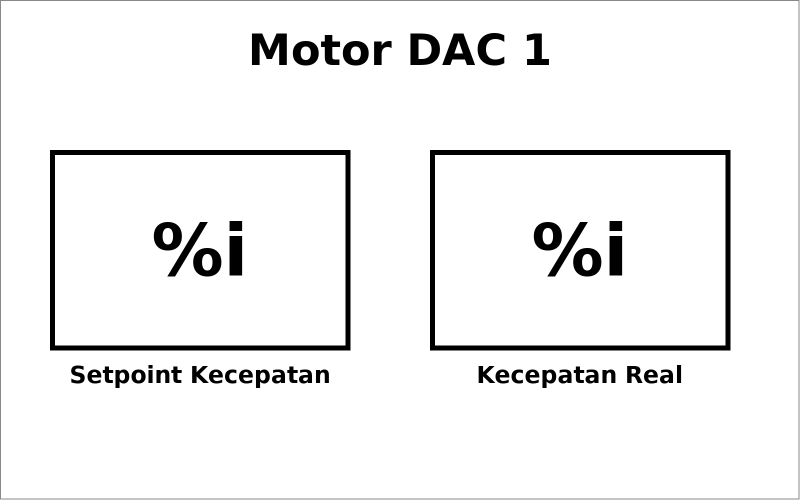
VISUALIZATION Screen_2_Sub_2  // 800x500
    Label (0,0 800x100), "Motor DAC 1"
    Rectangle (50,150 300x200), "%i", text variable: GVL.HMI_Motor_DAC_1_Input
        OnMouseClick: write GVL.HMI_Motor_DAC_1_Input via VisuDialogs.Numpad
    Label (50,350 300x50), "Setpoint Kecepatan"
    Label (430,350 300x50), "Kecepatan Real"
    Rectangle (430,150 300x200), "%i", text variable: GVL.HMI_Motor_DAC_1_Real
END_VISUALIZATION

(* stored: Version 1.1.0.1, ProductVersion 3.1.4024.12
   Visu Screen_2_Sub_2: Id {135a9eb4-6e55-44eb-83a0-2329cd818bb6} *)
